TYPE WinderParam_Typ :
STRUCT
	
	CalculatedRotSpeed:LREAL;
	CalculatedGear:LREAL;
	Tension:Tension_Typ;

END_STRUCT
END_TYPE

(* stored: Version 1.1.0.1, ProductVersion 3.1.4024.3
   DUT WinderParam_Typ: Id {417761dc-7b5c-4499-a4a4-411ac08562f8} *)
